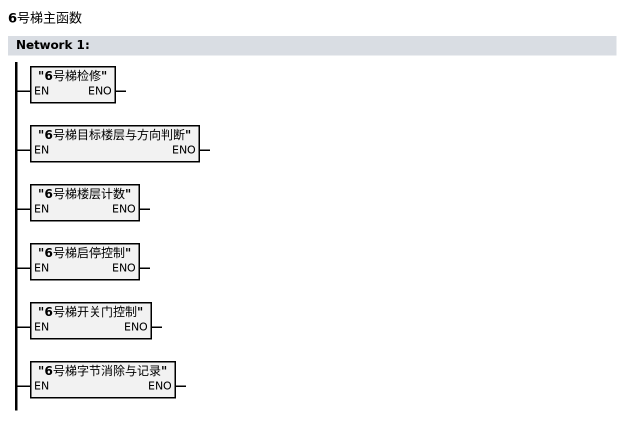
   RUNG wire#powerrail
      "6号梯检修"()
   END_RUNG
   RUNG wire#powerrail
      "6号梯目标楼层与方向判断"()
   END_RUNG
   RUNG wire#powerrail
      "6号梯楼层计数"()
   END_RUNG
   RUNG wire#powerrail
      "6号梯启停控制"()
   END_RUNG
   RUNG wire#powerrail
      "6号梯开关门控制"()
   END_RUNG
   RUNG wire#powerrail
      "6号梯字节消除与记录"()
   END_RUNG
   // the same network as SCL:
   "6号梯检修"();
   "6号梯目标楼层与方向判断"();
   "6号梯楼层计数"();
   "6号梯启停控制"();
   "6号梯开关门控制"();
   "6号梯字节消除与记录"();
END_REGION
END_FUNCTION

FUNCTION "6号梯运行监控模块" : Void   // FC19, LAD
{ S7_Optimized_Access := 'TRUE' }
VERSION : 0.1
BEGIN

REGION Network 1: 6号梯获取当前楼层设置标志位
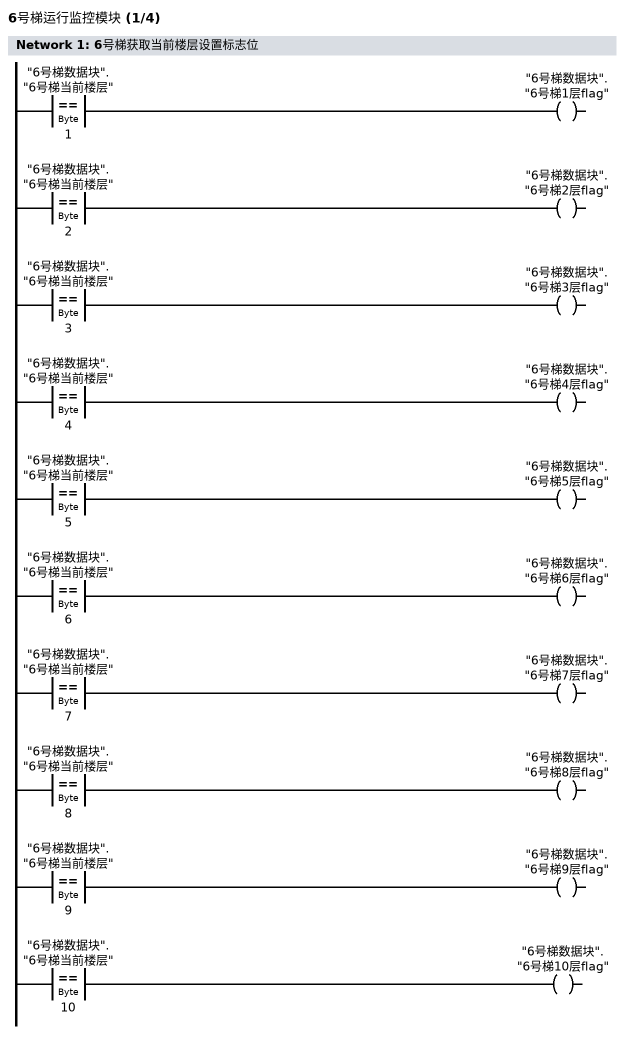
   RUNG wire#powerrail
      { S7_Templates := "SrcType := Byte" } EQ_Contact(in1 := "6号梯数据块"."6号梯当前楼层", in2 := 1)
      Coil( "6号梯数据块"."6号梯1层flag" )
   END_RUNG
   RUNG wire#powerrail
      { S7_Templates := "SrcType := Byte" } EQ_Contact(in1 := "6号梯数据块"."6号梯当前楼层", in2 := 2)
      Coil( "6号梯数据块"."6号梯2层flag" )
   END_RUNG
   RUNG wire#powerrail
      { S7_Templates := "SrcType := Byte" } EQ_Contact(in1 := "6号梯数据块"."6号梯当前楼层", in2 := 3)
      Coil( "6号梯数据块"."6号梯3层flag" )
   END_RUNG
   RUNG wire#powerrail
      { S7_Templates := "SrcType := Byte" } EQ_Contact(in1 := "6号梯数据块"."6号梯当前楼层", in2 := 4)
      Coil( "6号梯数据块"."6号梯4层flag" )
   END_RUNG
   RUNG wire#powerrail
      { S7_Templates := "SrcType := Byte" } EQ_Contact(in1 := "6号梯数据块"."6号梯当前楼层", in2 := 5)
      Coil( "6号梯数据块"."6号梯5层flag" )
   END_RUNG
   RUNG wire#powerrail
      { S7_Templates := "SrcType := Byte" } EQ_Contact(in1 := "6号梯数据块"."6号梯当前楼层", in2 := 6)
      Coil( "6号梯数据块"."6号梯6层flag" )
   END_RUNG
   RUNG wire#powerrail
      { S7_Templates := "SrcType := Byte" } EQ_Contact(in1 := "6号梯数据块"."6号梯当前楼层", in2 := 7)
      Coil( "6号梯数据块"."6号梯7层flag" )
   END_RUNG
   RUNG wire#powerrail
      { S7_Templates := "SrcType := Byte" } EQ_Contact(in1 := "6号梯数据块"."6号梯当前楼层", in2 := 8)
      Coil( "6号梯数据块"."6号梯8层flag" )
   END_RUNG
   RUNG wire#powerrail
      { S7_Templates := "SrcType := Byte" } EQ_Contact(in1 := "6号梯数据块"."6号梯当前楼层", in2 := 9)
      Coil( "6号梯数据块"."6号梯9层flag" )
   END_RUNG
   RUNG wire#powerrail
      { S7_Templates := "SrcType := Byte" } EQ_Contact(in1 := "6号梯数据块"."6号梯当前楼层", in2 := 10)
      Coil( "6号梯数据块"."6号梯10层flag" )
   END_RUNG
   // the same network as SCL:
   "6号梯数据块"."6号梯1层flag" := "6号梯数据块"."6号梯当前楼层" = 1;
   "6号梯数据块"."6号梯2层flag" := "6号梯数据块"."6号梯当前楼层" = 2;
   "6号梯数据块"."6号梯3层flag" := "6号梯数据块"."6号梯当前楼层" = 3;
   "6号梯数据块"."6号梯4层flag" := "6号梯数据块"."6号梯当前楼层" = 4;
   "6号梯数据块"."6号梯5层flag" := "6号梯数据块"."6号梯当前楼层" = 5;
   "6号梯数据块"."6号梯6层flag" := "6号梯数据块"."6号梯当前楼层" = 6;
   "6号梯数据块"."6号梯7层flag" := "6号梯数据块"."6号梯当前楼层" = 7;
   "6号梯数据块"."6号梯8层flag" := "6号梯数据块"."6号梯当前楼层" = 8;
   "6号梯数据块"."6号梯9层flag" := "6号梯数据块"."6号梯当前楼层" = 9;
   "6号梯数据块"."6号梯10层flag" := "6号梯数据块"."6号梯当前楼层" = 10;
END_REGION

REGION Network 2: 6号梯楼层led_a显示
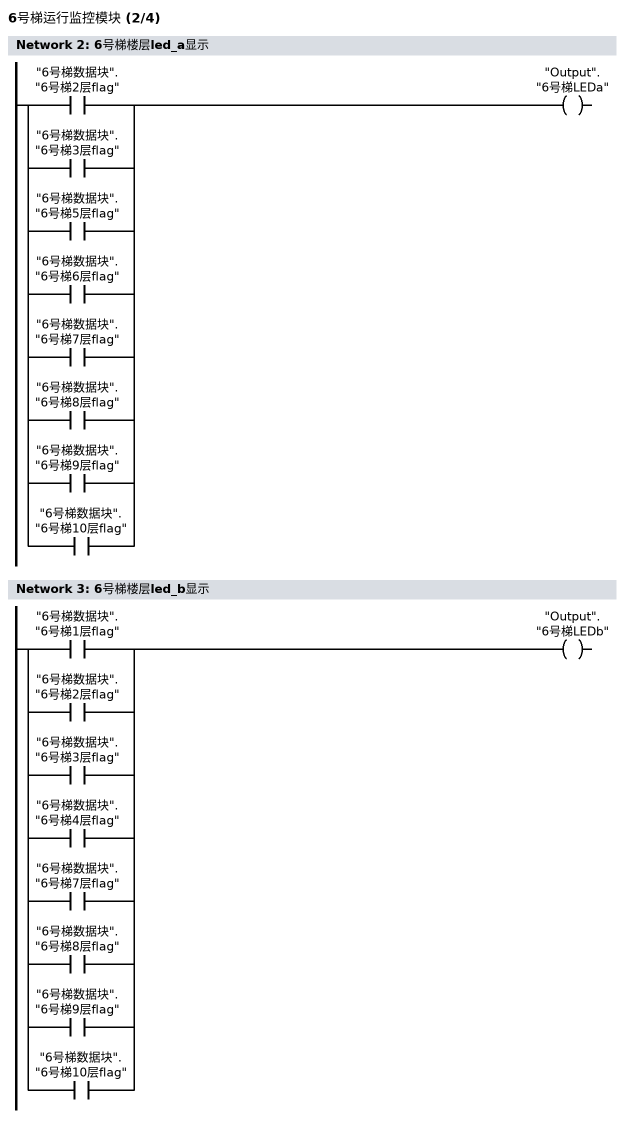
   RUNG wire#powerrail
      Contact( "6号梯数据块"."6号梯2层flag" )
      wire#w1
      Coil( "Output"."6号梯LEDa" )
   END_RUNG
   RUNG wire#powerrail
      Contact( "6号梯数据块"."6号梯3层flag" )
   END_RUNG wire#w1
   RUNG wire#powerrail
      Contact( "6号梯数据块"."6号梯5层flag" )
   END_RUNG wire#w1
   RUNG wire#powerrail
      Contact( "6号梯数据块"."6号梯6层flag" )
   END_RUNG wire#w1
   RUNG wire#powerrail
      Contact( "6号梯数据块"."6号梯7层flag" )
   END_RUNG wire#w1
   RUNG wire#powerrail
      Contact( "6号梯数据块"."6号梯8层flag" )
   END_RUNG wire#w1
   RUNG wire#powerrail
      Contact( "6号梯数据块"."6号梯9层flag" )
   END_RUNG wire#w1
   RUNG wire#powerrail
      Contact( "6号梯数据块"."6号梯10层flag" )
   END_RUNG wire#w1
   // the same network as SCL:
   "Output"."6号梯LEDa" := "6号梯数据块"."6号梯2层flag" OR "6号梯数据块"."6号梯3层flag" OR "6号梯数据块"."6号梯5层flag" OR "6号梯数据块"."6号梯6层flag" OR "6号梯数据块"."6号梯7层flag" OR "6号梯数据块"."6号梯8层flag" OR "6号梯数据块"."6号梯9层flag" OR "6号梯数据块"."6号梯10层flag";
END_REGION

REGION Network 3: 6号梯楼层led_b显示
   RUNG wire#powerrail
      Contact( "6号梯数据块"."6号梯1层flag" )
      wire#w1
      Coil( "Output"."6号梯LEDb" )
   END_RUNG
   RUNG wire#powerrail
      Contact( "6号梯数据块"."6号梯2层flag" )
   END_RUNG wire#w1
   RUNG wire#powerrail
      Contact( "6号梯数据块"."6号梯3层flag" )
   END_RUNG wire#w1
   RUNG wire#powerrail
      Contact( "6号梯数据块"."6号梯4层flag" )
   END_RUNG wire#w1
   RUNG wire#powerrail
      Contact( "6号梯数据块"."6号梯7层flag" )
   END_RUNG wire#w1
   RUNG wire#powerrail
      Contact( "6号梯数据块"."6号梯8层flag" )
   END_RUNG wire#w1
   RUNG wire#powerrail
      Contact( "6号梯数据块"."6号梯9层flag" )
   END_RUNG wire#w1
   RUNG wire#powerrail
      Contact( "6号梯数据块"."6号梯10层flag" )
   END_RUNG wire#w1
   // the same network as SCL:
   "Output"."6号梯LEDb" := "6号梯数据块"."6号梯1层flag" OR "6号梯数据块"."6号梯2层flag" OR "6号梯数据块"."6号梯3层flag" OR "6号梯数据块"."6号梯4层flag" OR "6号梯数据块"."6号梯7层flag" OR "6号梯数据块"."6号梯8层flag" OR "6号梯数据块"."6号梯9层flag" OR "6号梯数据块"."6号梯10层flag";
END_REGION

REGION Network 4: 6号梯楼层led_c显示
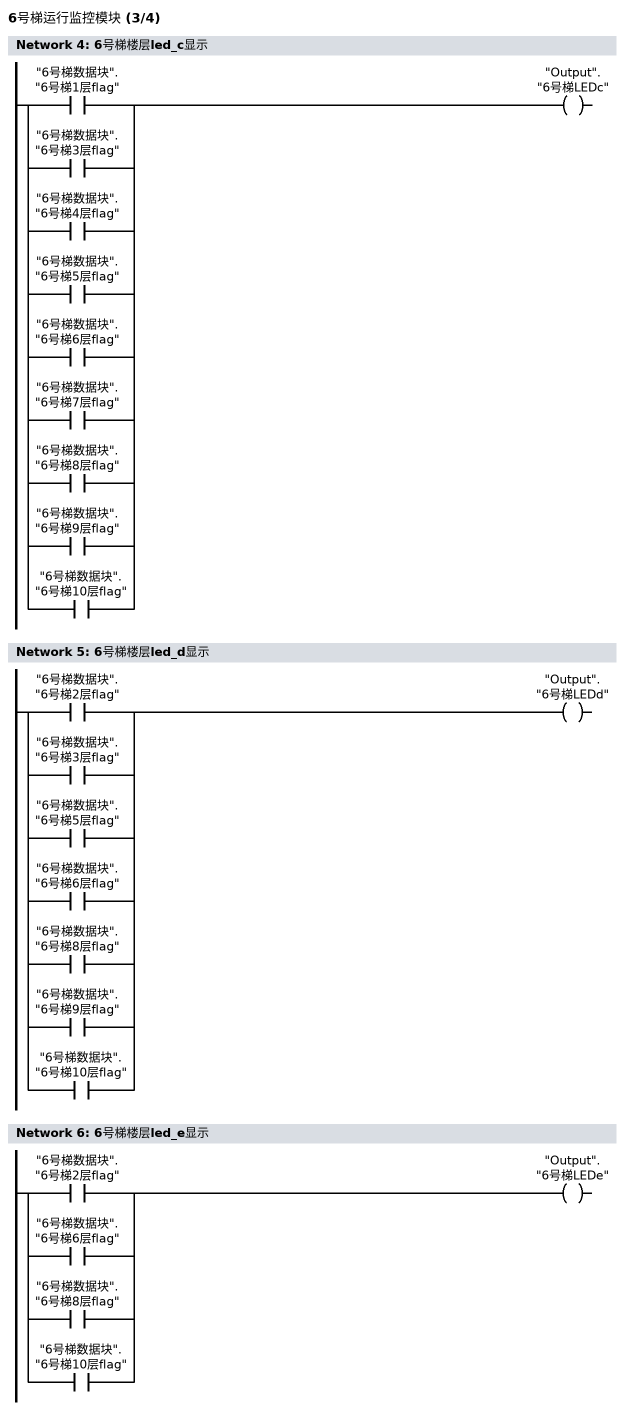
   RUNG wire#powerrail
      Contact( "6号梯数据块"."6号梯1层flag" )
      wire#w1
      Coil( "Output"."6号梯LEDc" )
   END_RUNG
   RUNG wire#powerrail
      Contact( "6号梯数据块"."6号梯3层flag" )
   END_RUNG wire#w1
   RUNG wire#powerrail
      Contact( "6号梯数据块"."6号梯4层flag" )
   END_RUNG wire#w1
   RUNG wire#powerrail
      Contact( "6号梯数据块"."6号梯5层flag" )
   END_RUNG wire#w1
   RUNG wire#powerrail
      Contact( "6号梯数据块"."6号梯6层flag" )
   END_RUNG wire#w1
   RUNG wire#powerrail
      Contact( "6号梯数据块"."6号梯7层flag" )
   END_RUNG wire#w1
   RUNG wire#powerrail
      Contact( "6号梯数据块"."6号梯8层flag" )
   END_RUNG wire#w1
   RUNG wire#powerrail
      Contact( "6号梯数据块"."6号梯9层flag" )
   END_RUNG wire#w1
   RUNG wire#powerrail
      Contact( "6号梯数据块"."6号梯10层flag" )
   END_RUNG wire#w1
   // the same network as SCL:
   "Output"."6号梯LEDc" := "6号梯数据块"."6号梯1层flag" OR "6号梯数据块"."6号梯3层flag" OR "6号梯数据块"."6号梯4层flag" OR "6号梯数据块"."6号梯5层flag" OR "6号梯数据块"."6号梯6层flag" OR "6号梯数据块"."6号梯7层flag" OR "6号梯数据块"."6号梯8层flag" OR "6号梯数据块"."6号梯9层flag" OR "6号梯数据块"."6号梯10层flag";
END_REGION

REGION Network 5: 6号梯楼层led_d显示
   RUNG wire#powerrail
      Contact( "6号梯数据块"."6号梯2层flag" )
      wire#w1
      Coil( "Output"."6号梯LEDd" )
   END_RUNG
   RUNG wire#powerrail
      Contact( "6号梯数据块"."6号梯3层flag" )
   END_RUNG wire#w1
   RUNG wire#powerrail
      Contact( "6号梯数据块"."6号梯5层flag" )
   END_RUNG wire#w1
   RUNG wire#powerrail
      Contact( "6号梯数据块"."6号梯6层flag" )
   END_RUNG wire#w1
   RUNG wire#powerrail
      Contact( "6号梯数据块"."6号梯8层flag" )
   END_RUNG wire#w1
   RUNG wire#powerrail
      Contact( "6号梯数据块"."6号梯9层flag" )
   END_RUNG wire#w1
   RUNG wire#powerrail
      Contact( "6号梯数据块"."6号梯10层flag" )
   END_RUNG wire#w1
   // the same network as SCL:
   "Output"."6号梯LEDd" := "6号梯数据块"."6号梯2层flag" OR "6号梯数据块"."6号梯3层flag" OR "6号梯数据块"."6号梯5层flag" OR "6号梯数据块"."6号梯6层flag" OR "6号梯数据块"."6号梯8层flag" OR "6号梯数据块"."6号梯9层flag" OR "6号梯数据块"."6号梯10层flag";
END_REGION

REGION Network 6: 6号梯楼层led_e显示
   RUNG wire#powerrail
      Contact( "6号梯数据块"."6号梯2层flag" )
      wire#w1
      Coil( "Output"."6号梯LEDe" )
   END_RUNG
   RUNG wire#powerrail
      Contact( "6号梯数据块"."6号梯6层flag" )
   END_RUNG wire#w1
   RUNG wire#powerrail
      Contact( "6号梯数据块"."6号梯8层flag" )
   END_RUNG wire#w1
   RUNG wire#powerrail
      Contact( "6号梯数据块"."6号梯10层flag" )
   END_RUNG wire#w1
   // the same network as SCL:
   "Output"."6号梯LEDe" := "6号梯数据块"."6号梯2层flag" OR "6号梯数据块"."6号梯6层flag" OR "6号梯数据块"."6号梯8层flag" OR "6号梯数据块"."6号梯10层flag";
END_REGION

REGION Network 7: 6号梯楼层led_f显示
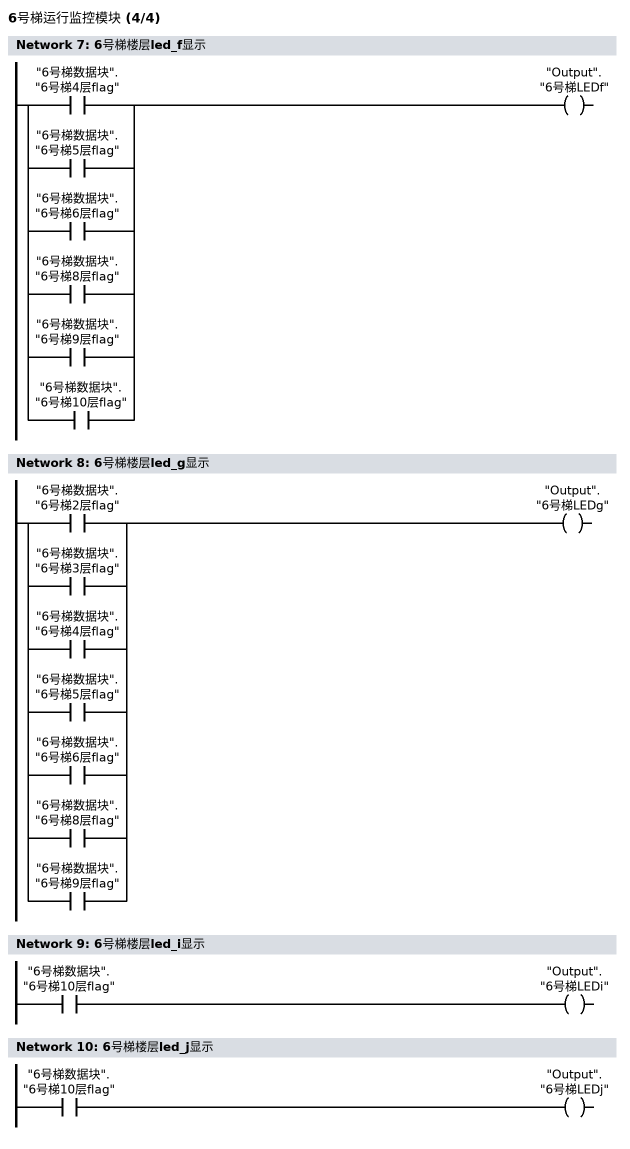
   RUNG wire#powerrail
      Contact( "6号梯数据块"."6号梯4层flag" )
      wire#w1
      Coil( "Output"."6号梯LEDf" )
   END_RUNG
   RUNG wire#powerrail
      Contact( "6号梯数据块"."6号梯5层flag" )
   END_RUNG wire#w1
   RUNG wire#powerrail
      Contact( "6号梯数据块"."6号梯6层flag" )
   END_RUNG wire#w1
   RUNG wire#powerrail
      Contact( "6号梯数据块"."6号梯8层flag" )
   END_RUNG wire#w1
   RUNG wire#powerrail
      Contact( "6号梯数据块"."6号梯9层flag" )
   END_RUNG wire#w1
   RUNG wire#powerrail
      Contact( "6号梯数据块"."6号梯10层flag" )
   END_RUNG wire#w1
   // the same network as SCL:
   "Output"."6号梯LEDf" := "6号梯数据块"."6号梯4层flag" OR "6号梯数据块"."6号梯5层flag" OR "6号梯数据块"."6号梯6层flag" OR "6号梯数据块"."6号梯8层flag" OR "6号梯数据块"."6号梯9层flag" OR "6号梯数据块"."6号梯10层flag";
END_REGION

REGION Network 8: 6号梯楼层led_g显示
   RUNG wire#powerrail
      Contact( "6号梯数据块"."6号梯2层flag" )
      wire#w1
      Coil( "Output"."6号梯LEDg" )
   END_RUNG
   RUNG wire#powerrail
      Contact( "6号梯数据块"."6号梯3层flag" )
   END_RUNG wire#w1
   RUNG wire#powerrail
      Contact( "6号梯数据块"."6号梯4层flag" )
   END_RUNG wire#w1
   RUNG wire#powerrail
      Contact( "6号梯数据块"."6号梯5层flag" )
   END_RUNG wire#w1
   RUNG wire#powerrail
      Contact( "6号梯数据块"."6号梯6层flag" )
   END_RUNG wire#w1
   RUNG wire#powerrail
      Contact( "6号梯数据块"."6号梯8层flag" )
   END_RUNG wire#w1
   RUNG wire#powerrail
      Contact( "6号梯数据块"."6号梯9层flag" )
   END_RUNG wire#w1
   // the same network as SCL:
   "Output"."6号梯LEDg" := "6号梯数据块"."6号梯2层flag" OR "6号梯数据块"."6号梯3层flag" OR "6号梯数据块"."6号梯4层flag" OR "6号梯数据块"."6号梯5层flag" OR "6号梯数据块"."6号梯6层flag" OR "6号梯数据块"."6号梯8层flag" OR "6号梯数据块"."6号梯9层flag";
END_REGION

REGION Network 9: 6号梯楼层led_i显示
   RUNG wire#powerrail
      Contact( "6号梯数据块"."6号梯10层flag" )
      Coil( "Output"."6号梯LEDi" )
   END_RUNG
   // the same network as SCL:
   "Output"."6号梯LEDi" := "6号梯数据块"."6号梯10层flag";
END_REGION

REGION Network 10: 6号梯楼层led_j显示
   RUNG wire#powerrail
      Contact( "6号梯数据块"."6号梯10层flag" )
      Coil( "Output"."6号梯LEDj" )
   END_RUNG
   // the same network as SCL:
   "Output"."6号梯LEDj" := "6号梯数据块"."6号梯10层flag";
END_REGION
END_FUNCTION

FUNCTION "6号梯超重与内选" : Void   // FC25, LAD
{ S7_Optimized_Access := 'TRUE' }
VERSION : 0.1
BEGIN
END_FUNCTION

FUNCTION "6号梯开关门控制" : Void   // FC31, LAD
{ S7_Optimized_Access := 'TRUE' }
VERSION : 0.1
BEGIN
END_FUNCTION

FUNCTION "6号梯楼层计数" : Void   // FC37, LAD
{ S7_Optimized_Access := 'TRUE' }
VERSION : 0.1
BEGIN
END_FUNCTION

FUNCTION "6号梯检修" : Void   // FC56, LAD
{ S7_Optimized_Access := 'TRUE' }
VERSION : 0.1
BEGIN
END_FUNCTION

FUNCTION "6号梯目标楼层与方向判断" : Void   // FC57, LAD
{ S7_Optimized_Access := 'TRUE' }
VERSION : 0.1
BEGIN
END_FUNCTION

FUNCTION "6号梯字节消除与记录" : Void   // FC58, LAD
{ S7_Optimized_Access := 'TRUE' }
VERSION : 0.1
BEGIN
END_FUNCTION

FUNCTION "6号梯启停控制" : Void   // FC63, LAD
{ S7_Optimized_Access := 'TRUE' }
VERSION : 0.1
BEGIN
END_FUNCTION

// folder: 群控算法

FUNCTION "群控算法" : Void   // FC38, SCL
{ S7_Optimized_Access := 'TRUE' }
VERSION : 0.1
BEGIN
END_FUNCTION

// folder: 群控算法/电梯算法

FUNCTION "体重转换" : Void   // FC40, LAD
{ S7_Optimized_Access := 'TRUE' }
VERSION : 0.1
   VAR_INPUT
      in : Word;
   END_VAR
   VAR_OUTPUT
      out : Word;
   END_VAR
   VAR_TEMP
      temp : Real;
   END_VAR
BEGIN

REGION Network 1: 体重转换
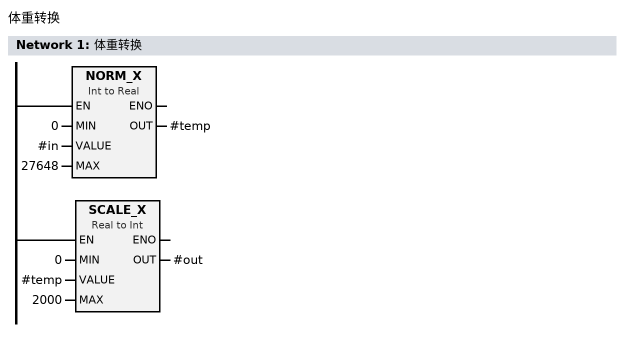
   RUNG wire#powerrail
      { S7_Templates := "[SrcType := Int, DestType := Real]" } Normalize(min := 0, value := #in, max := 27648, out => #temp)
   END_RUNG
   RUNG wire#powerrail
      { S7_Templates := "[SrcType := Real, DestType := Int]" } Scale(min := 0, value := #temp, max := 2000, out => #out)
   END_RUNG
   // the same network as SCL:
   #temp := NORM_X(MIN := 0, VALUE := #in, MAX := 27648);
   #out := SCALE_X(MIN := 0, VALUE := #temp, MAX := 2000);
END_REGION
END_FUNCTION